PROGRAM P2_05_Process_Ctrl
VAR
	bWaitAferBatchClose			:BOOL;
	tonWaitAfterBatchClose		:TON;
	tonMixerDelayStopped: TON;
END_VAR
VAR // added by the converter: edge detectors and wires of the graphical bodies
    _w1, _w2, _w3 : BOOL;
    _rt1 : R_TRIG;
END_VAR

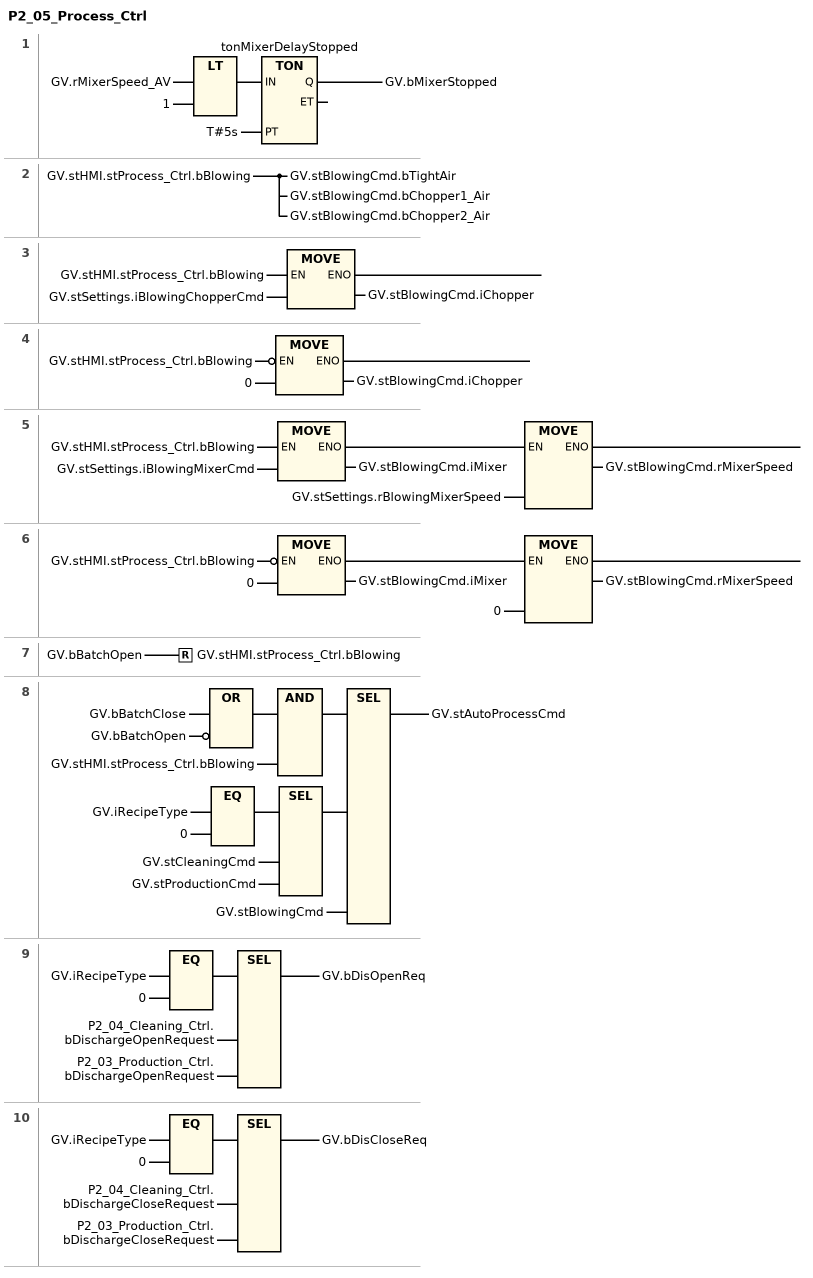
// NETWORK 1
tonMixerDelayStopped(IN := GV.rMixerSpeed_AV < 1, PT := T#5s); // TON
GV.bMixerStopped := tonMixerDelayStopped.Q;

// NETWORK 2
_w1 := GV.stHMI.stProcess_Ctrl.bBlowing;
GV.stBlowingCmd.bTightAir := _w1;
GV.stBlowingCmd.bChopper1_Air := _w1;
GV.stBlowingCmd.bChopper2_Air := _w1;

// NETWORK 3
IF GV.stHMI.stProcess_Ctrl.bBlowing THEN GV.stBlowingCmd.iChopper := GV.stSettings.iBlowingChopperCmd; END_IF

// NETWORK 4
IF NOT GV.stHMI.stProcess_Ctrl.bBlowing THEN GV.stBlowingCmd.iChopper := 0; END_IF

// NETWORK 5
_w2 := GV.stHMI.stProcess_Ctrl.bBlowing;
IF _w2 THEN GV.stBlowingCmd.iMixer := GV.stSettings.iBlowingMixerCmd; END_IF
IF _w2 THEN GV.stBlowingCmd.rMixerSpeed := GV.stSettings.rBlowingMixerSpeed; END_IF

// NETWORK 6
_w3 := NOT GV.stHMI.stProcess_Ctrl.bBlowing;
IF _w3 THEN GV.stBlowingCmd.iMixer := 0; END_IF
IF _w3 THEN GV.stBlowingCmd.rMixerSpeed := 0; END_IF

// NETWORK 7
GV.stHMI.stProcess_Ctrl.bBlowing R= GV.bBatchOpen;

// NETWORK 8
GV.stAutoProcessCmd := SEL((GV.bBatchClose OR NOT GV.bBatchOpen) AND GV.stHMI.stProcess_Ctrl.bBlowing, SEL(GV.iRecipeType = 0, GV.stCleaningCmd, GV.stProductionCmd), GV.stBlowingCmd);

// NETWORK 9
GV.bDisOpenReq := SEL(GV.iRecipeType = 0, P2_04_Cleaning_Ctrl.bDischargeOpenRequest, P2_03_Production_Ctrl.bDischargeOpenRequest);

// NETWORK 10
GV.bDisCloseReq := SEL(GV.iRecipeType = 0, P2_04_Cleaning_Ctrl.bDischargeCloseRequest, P2_03_Production_Ctrl.bDischargeCloseRequest);

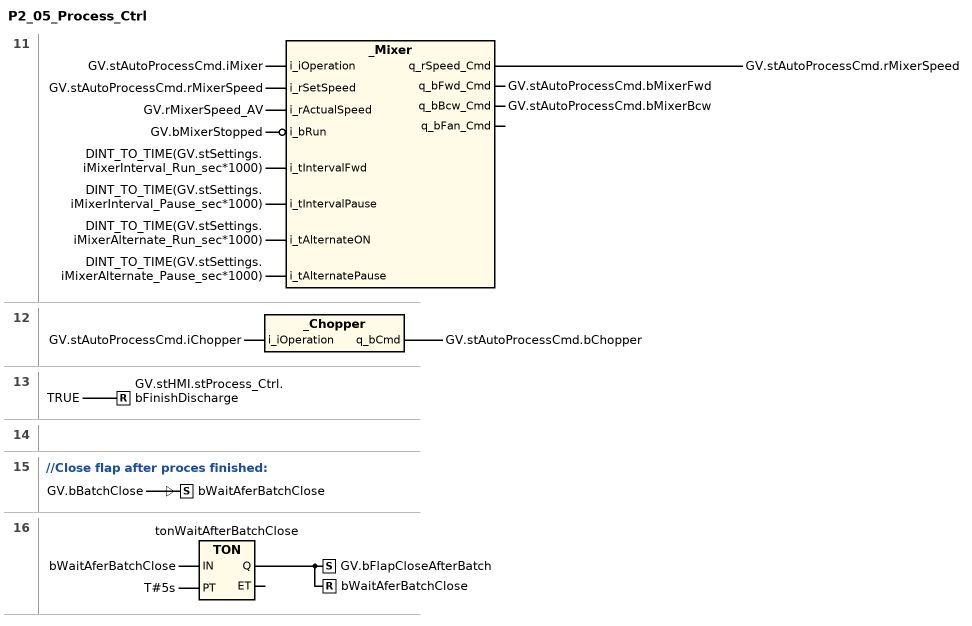
// NETWORK 11
_Mixer(i_iOperation := GV.stAutoProcessCmd.iMixer, i_rSetSpeed := GV.stAutoProcessCmd.rMixerSpeed, i_rActualSpeed := GV.rMixerSpeed_AV, i_bRun := NOT GV.bMixerStopped, i_tIntervalFwd := DINT_TO_TIME(GV.stSettings.iMixerInterval_Run_sec*1000), i_tIntervalPause := DINT_TO_TIME(GV.stSettings.iMixerInterval_Pause_sec*1000), i_tAlternateON := DINT_TO_TIME(GV.stSettings.iMixerAlternate_Run_sec*1000), i_tAlternatePause := DINT_TO_TIME(GV.stSettings.iMixerAlternate_Pause_sec*1000), q_bFwd_Cmd => GV.stAutoProcessCmd.bMixerFwd, q_bBcw_Cmd => GV.stAutoProcessCmd.bMixerBcw);
GV.stAutoProcessCmd.rMixerSpeed := _Mixer.q_rSpeed_Cmd;

// NETWORK 12
_Chopper(i_iOperation := GV.stAutoProcessCmd.iChopper);
GV.stAutoProcessCmd.bChopper := _Chopper.q_bCmd;

// NETWORK 13
GV.stHMI.stProcess_Ctrl.bFinishDischarge R= TRUE;

// NETWORK 14

// NETWORK 15
// label: //Close flap after proces finished
_rt1(CLK := GV.bBatchClose);
bWaitAferBatchClose S= _rt1.Q;

// NETWORK 16
tonWaitAfterBatchClose(IN := bWaitAferBatchClose, PT := T#5s); // TON
GV.bFlapCloseAfterBatch S= tonWaitAfterBatchClose.Q;
bWaitAferBatchClose R= tonWaitAfterBatchClose.Q;

END_PROGRAM

(* stored: Version 1.1.0.1
   POU P2_05_Process_Ctrl: Id {e867a8fd-57c7-4ddf-9933-795cf451023c}, SpecialFunc None *)
